// TIA Portal V18 export
TYPE "LGasp_type_Prg_Impilaggio"
// stored: IsFailsafeCompliant false
   STRUCT
      nomeprogramma : WString[30];   // nome del programma trasferito dal PC
      ID : DInt;   // ID programma
      Tipoimpilaggio : DInt;   // valore numerico da definire in base alla commessa
      DeltaX : LReal;   // [mm] incremento in X fra colonne adiacenti
      DeltaY : LReal;   // [mm] incremento in Y fra colonne adiacenti (solo in caso di colonne in 2 dimensioni)
      DeltaZ : LReal;   // [mm] incremento in Z fra righe adiacenti
      NrPzMaxPacco : DInt;   // Numero massimo di pezzi del pacco
      X_MaxPacco : LReal;   // [mm] Larghezza X massima del pacco
      Y_MaxPacco : LReal;   // [mm] Larghezza Y massima del pacco (solo in caso di colonne in 2 dimensioni)
      Z_MaxPacco : LReal;   // [mm] Altezza Z massima del pacco
      PesoTotMaxPacco : LReal;   // [kg] Peso totale massimo del pacco
      PesoLineareMaxPacco : LReal;   // [kg/m] Peso massimo del pacco per metro di lunghezza (opzionale)
      Opzioni : Array[1..16] of Bool;   // opzioni varie (modalità di impilaggio, film ecc..)
      Opzione1 : Int;   // opzioni varie disponibili
      Opzione2 : String;   // opzioni varie disponibili
      Opzione3 : Real;   // opzioni varie disponibili
      Correttori : Array[1..20] of LReal;   // correttori disponibili per funzioni varie
      Limiti : Struct
         DeltaX_min : LReal := -730.0;   // Valore minimo impostabile da HMI
         DeltaX_max : LReal := 730.0;   // Valore massimo impostabile da HMI
         DeltaY_min : LReal;   // Valore minimo impostabile da HMI
         DeltaY_max : LReal;   // Valore massimo impostabile da HMI
         DeltaZ_min : LReal := 0.0;   // Valore minimo impostabile da HMI
         DeltaZ_max : LReal := 50.0;   // Valore massimo impostabile da HMI
         NrPzMaxPacco_min : DInt := 1;   // Valore minimo impostabile da HMI
         NrPzMaxPacco_max : DInt := 10000;   // Valore massimo impostabile da HMI
         X_MaxPacco_min : LReal := 0.0;   // Valore minimo impostabile da HMI
         X_MaxPacco_max : LReal := 730.0;   // Valore massimo impostabile da HMI
         Y_MaxPacco_min : LReal := 0.0;   // Valore minimo impostabile da HMI
         Y_MaxPacco_max : LReal := 6000.0;   // Valore massimo impostabile da HMI
         Z_MaxPacco_min : LReal := 0.0;   // Valore minimo impostabile da HMI
         Z_MaxPacco_max : LReal := 600.0;   // Valore massimo impostabile da HMI
         PesoTotMaxPacco_min : LReal := 0.0;   // Valore minimo impostabile da HMI
         PesoTotMaxPacco_max : LReal := 3000.0;   // Valore massimo impostabile da HMI
         PesoLineareMaxPacco_min : LReal := 0.0;   // Valore minimo impostabile da HMI
         PesoLineareMaxPacco_max : LReal := 3000.0;   // Valore massimo impostabile da HMI
      END_STRUCT;
   END_STRUCT;
   // // Opzioni[1] : Presenza cartone 1=si
   // // Opzioni[2] : Presenza reggie 1=si
   // // Opzioni[3] : Presenza film 1=si
END_TYPE
